// Mitsubishi GX Works2 project: SEQUENCE_REPEAT_DANSOK   PLC: Q03UDV

PROGRAM MAIN
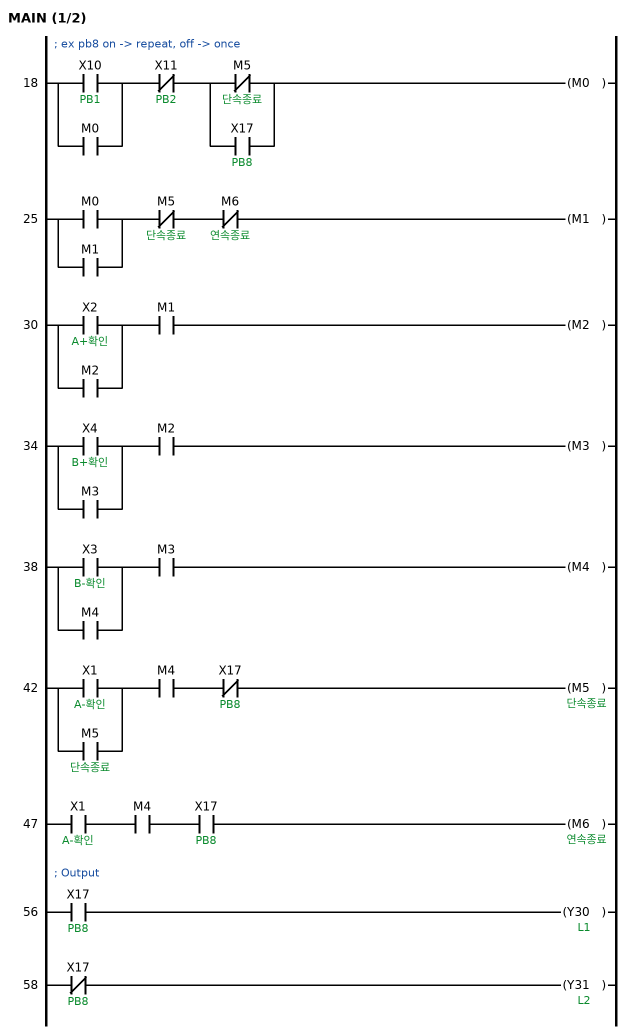
; ex pb8 on -> repeat, off -> once
18    LD      X10  ; PB1
      OR      M0
      ANI     X11  ; PB2
      LDI     M5  ; 단속종료
      OR      X17  ; PB8
      ANB
      OUT     M0
25    LD      M0
      OR      M1
      ANI     M5  ; 단속종료
      ANI     M6  ; 연속종료
      OUT     M1
30    LD      X2  ; A+확인
      OR      M2
      AND     M1
      OUT     M2
34    LD      X4  ; B+확인
      OR      M3
      AND     M2
      OUT     M3
38    LD      X3  ; B-확인
      OR      M4
      AND     M3
      OUT     M4
42    LD      X1  ; A-확인
      OR      M5  ; 단속종료
      AND     M4
      ANI     X17  ; PB8
      OUT     M5  ; 단속종료
47    LD      X1  ; A-확인
      AND     M4
      AND     X17  ; PB8
      OUT     M6  ; 연속종료
; Output
56    LD      X17  ; PB8
      OUT     Y30  ; L1
58    LDI     X17  ; PB8
      OUT     Y31  ; L2
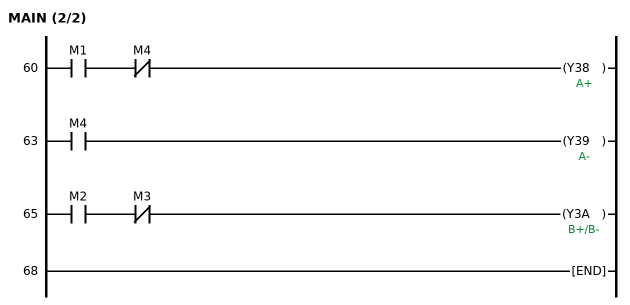
60    LD      M1
      ANI     M4
      OUT     Y38  ; A+
63    LD      M4
      OUT     Y39  ; A-
65    LD      M2
      ANI     M3
      OUT     Y3A  ; B+/B-
68    END
END_PROGRAM
